TYPE "UDT_LogEntry"
STRUCT
    stamp : DTL;
    value : Real;
END_STRUCT
END_TYPE
